// TIA Portal V20 export
FUNCTION_BLOCK "LER_AlignSyncMove"   // FB99, LAD
// stored: Access Published, MemoryReserve 100, SetENOAutomatically false
   VAR_INPUT
      enable : Bool;
      Anode : Bool;
      Cathode : Bool;
      AxisXHomePos { ExternalAccessible := 'False'; ExternalVisible := 'False'; ExternalWritable := 'False'} : LReal;
      AxisY1HomePos { ExternalAccessible := 'False'; ExternalVisible := 'False'; ExternalWritable := 'False'} : LReal;
      AxisY2HomePos { ExternalAccessible := 'False'; ExternalVisible := 'False'; ExternalWritable := 'False'} : LReal;
      MoveSpeed : LReal;
   END_VAR
   VAR_OUTPUT
      error : Bool;
      busy : Bool;
      done : Bool;
      status : Word;
   END_VAR
   VAR_IN_OUT
      moduleInterface : "LER_typeAlignSyncMoveInterface";
      AlignTableAxisX : DB_ANY;
      AlignTableAxisY1 : DB_ANY;
      AlignTableAxisY2 : DB_ANY;
   END_VAR
   VAR
      statMoveRad : LReal;
      statThetaX_Rad : LReal;
      statThetaY1_Rad : LReal;
      statThetaY2_Rad : LReal;
      statDetlaX : LReal;
      statDetlaY1 : LReal;
      statDetlaY2 : LReal;
      instAlignTableAxisXMCMoveAbs : MC_MOVEABSOLUTE;
      instAlignTableAxisY1MCMoveAbs { S7_SetPoint := 'True'} : MC_MOVEABSOLUTE;
      instAlignTableAxisY2MCMoveAbs { S7_SetPoint := 'True'} : MC_MOVEABSOLUTE;
      statPulse { S7_SetPoint := 'True'} : Array[1..50] of Bool;
      statMoveXCmd : Array[1..10] of Bool;
      statMoveY1Cmd : Array[1..10] of Bool;
      statMoveY2Cmd : Array[1..10] of Bool;
   END_VAR
   VAR_TEMP
      tempAlignTableAxisX : REF_TO TO_SynchronousAxis;
      tempAlignTableAxisY1 : REF_TO TO_SynchronousAxis;
      tempAlignTableAxisY2 : REF_TO TO_SynchronousAxis;
   END_VAR
   VAR CONSTANT
      PI : LReal := 3.14159265358979;
      INITIAL_RAD : LReal := 0.0;
      CENTERRADIUS : LReal := 120.0;
   END_VAR
   VAR_TEMP   // added for the SCL form of the ladder/FBD networks
      _w1 : Bool;
   END_VAR
BEGIN

REGION Network 1 (SCL): Axis Config
   #tempAlignTableAxisY1 ?= #AlignTableAxisY1;
   #tempAlignTableAxisY2 ?= #AlignTableAxisY2;
   // #tempAlignTableAxisX ?= #AlignTableAxisX;
END_REGION

REGION Network 2: Error Check
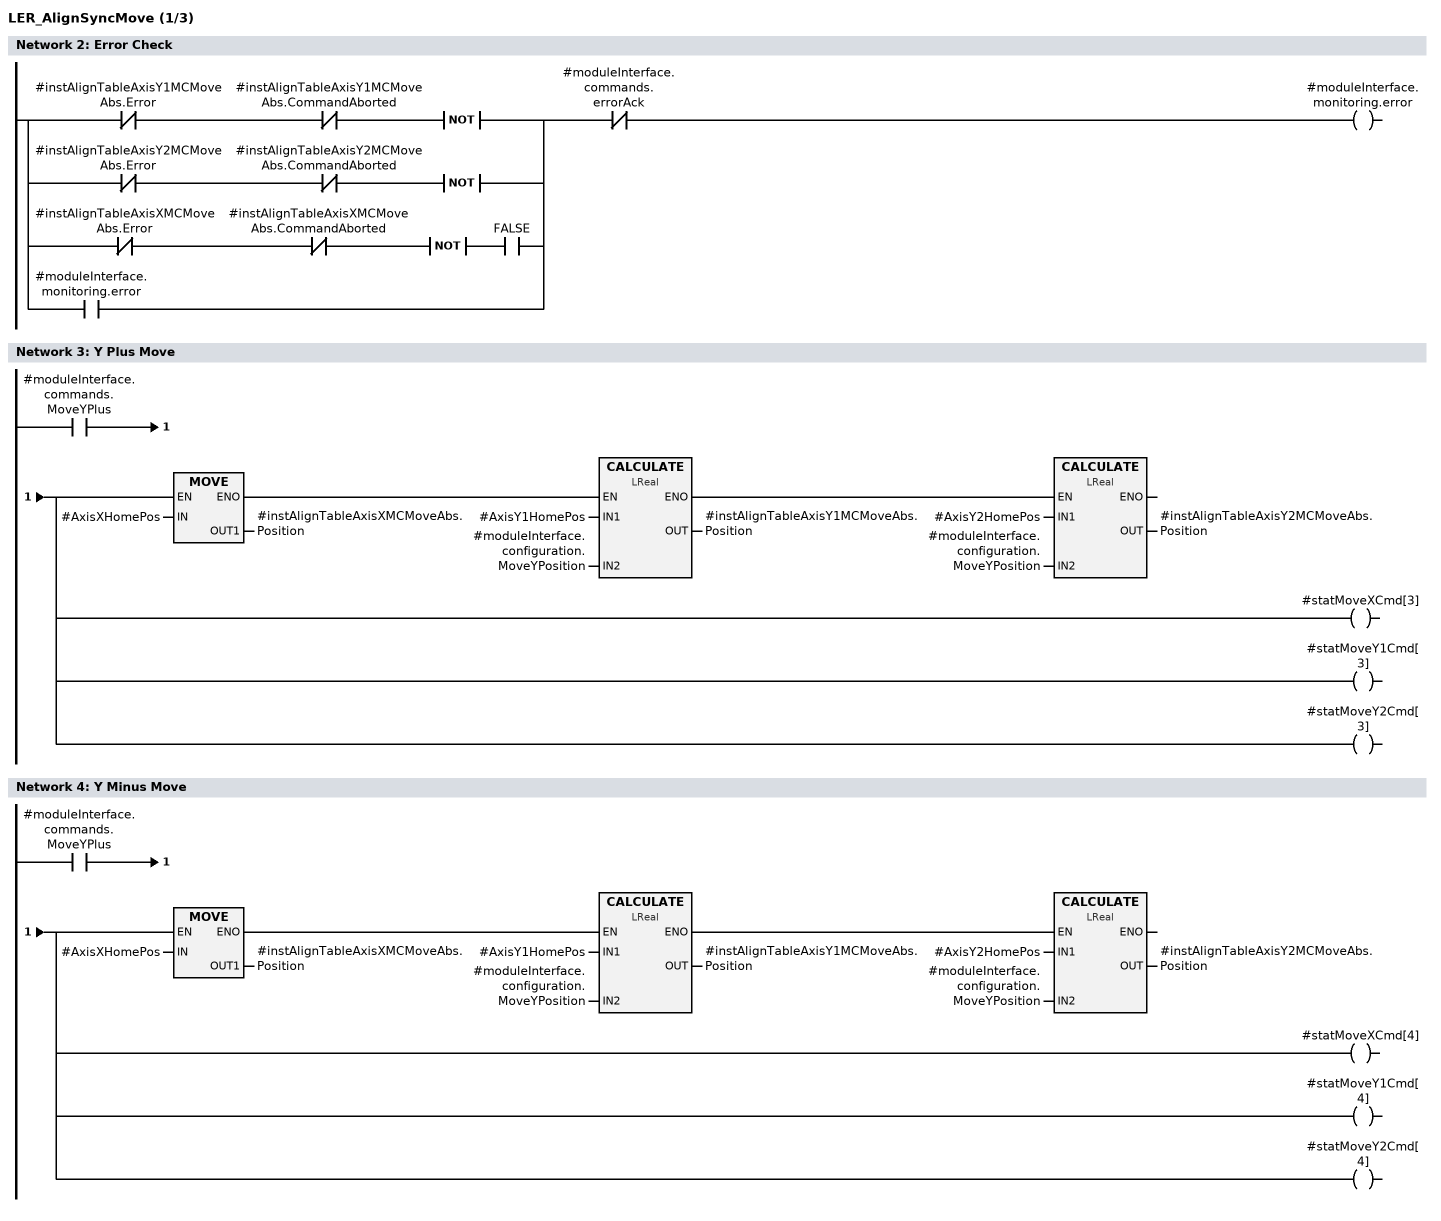
   RUNG wire#powerrail
      I_Contact( #instAlignTableAxisY1MCMoveAbs.Error )
      I_Contact( #instAlignTableAxisY1MCMoveAbs.CommandAborted )
      Not()
      wire#w1
      I_Contact( #moduleInterface.commands.errorAck )
      Coil( #moduleInterface.monitoring.error )
   END_RUNG
   RUNG wire#powerrail
      I_Contact( #instAlignTableAxisY2MCMoveAbs.Error )
      I_Contact( #instAlignTableAxisY2MCMoveAbs.CommandAborted )
      Not()
   END_RUNG wire#w1
   RUNG wire#powerrail
      I_Contact( #instAlignTableAxisXMCMoveAbs.Error )
      I_Contact( #instAlignTableAxisXMCMoveAbs.CommandAborted )
      Not()
      Contact( FALSE )
   END_RUNG wire#w1
   RUNG wire#powerrail
      Contact( #moduleInterface.monitoring.error )
   END_RUNG wire#w1
   // the same network as SCL:
   #moduleInterface.monitoring.error := (NOT (NOT #instAlignTableAxisY1MCMoveAbs.Error AND NOT #instAlignTableAxisY1MCMoveAbs.CommandAborted) OR NOT (NOT #instAlignTableAxisY2MCMoveAbs.Error AND NOT #instAlignTableAxisY2MCMoveAbs.CommandAborted) OR (NOT (NOT #instAlignTableAxisXMCMoveAbs.Error AND NOT #instAlignTableAxisXMCMoveAbs.CommandAborted) AND FALSE) OR #moduleInterface.monitoring.error) AND NOT #moduleInterface.commands.errorAck;
END_REGION

REGION Network 3: Y Plus Move
   RUNG wire#powerrail
      Contact( #moduleInterface.commands.MoveYPlus )
      wire#w1
      Move(in := #AxisXHomePos, out1 => #instAlignTableAxisXMCMoveAbs.Position)
      { S7_Templates := "SrcType := LReal"; S7_Expression := "IN1+IN2" } Calculate(in1 := #AxisY1HomePos, in2 := #moduleInterface.configuration.MoveYPosition, out => #instAlignTableAxisY1MCMoveAbs.Position)
      { S7_Templates := "SrcType := LReal"; S7_Expression := "IN1-IN2" } Calculate(in1 := #AxisY2HomePos, in2 := #moduleInterface.configuration.MoveYPosition, out => #instAlignTableAxisY2MCMoveAbs.Position)
   END_RUNG
   RUNG wire#w1
      Coil( #statMoveXCmd[3] )
   END_RUNG
   RUNG wire#w1
      Coil( #statMoveY1Cmd[3] )
   END_RUNG
   RUNG wire#w1
      Coil( #statMoveY2Cmd[3] )
   END_RUNG
   // the same network as SCL:
   IF #moduleInterface.commands.MoveYPlus THEN
       #instAlignTableAxisXMCMoveAbs.Position := #AxisXHomePos;
       #instAlignTableAxisY1MCMoveAbs.Position := #AxisY1HomePos+#moduleInterface.configuration.MoveYPosition;
       #instAlignTableAxisY2MCMoveAbs.Position := #AxisY2HomePos-#moduleInterface.configuration.MoveYPosition;
   END_IF;
   #statMoveXCmd[3] := #moduleInterface.commands.MoveYPlus;
   #statMoveY1Cmd[3] := #moduleInterface.commands.MoveYPlus;
   #statMoveY2Cmd[3] := #moduleInterface.commands.MoveYPlus;
END_REGION

REGION Network 4: Y Minus Move
   RUNG wire#powerrail
      Contact( #moduleInterface.commands.MoveYPlus )
      wire#w1
      Move(in := #AxisXHomePos, out1 => #instAlignTableAxisXMCMoveAbs.Position)
      { S7_Templates := "SrcType := LReal"; S7_Expression := "IN1-IN2" } Calculate(in1 := #AxisY1HomePos, in2 := #moduleInterface.configuration.MoveYPosition, out => #instAlignTableAxisY1MCMoveAbs.Position)
      { S7_Templates := "SrcType := LReal"; S7_Expression := "IN1+IN2" } Calculate(in1 := #AxisY2HomePos, in2 := #moduleInterface.configuration.MoveYPosition, out => #instAlignTableAxisY2MCMoveAbs.Position)
   END_RUNG
   RUNG wire#w1
      Coil( #statMoveXCmd[4] )
   END_RUNG
   RUNG wire#w1
      Coil( #statMoveY1Cmd[4] )
   END_RUNG
   RUNG wire#w1
      Coil( #statMoveY2Cmd[4] )
   END_RUNG
   // the same network as SCL:
   IF #moduleInterface.commands.MoveYPlus THEN
       #instAlignTableAxisXMCMoveAbs.Position := #AxisXHomePos;
       #instAlignTableAxisY1MCMoveAbs.Position := #AxisY1HomePos-#moduleInterface.configuration.MoveYPosition;
       #instAlignTableAxisY2MCMoveAbs.Position := #AxisY2HomePos+#moduleInterface.configuration.MoveYPosition;
   END_IF;
   #statMoveXCmd[4] := #moduleInterface.commands.MoveYPlus;
   #statMoveY1Cmd[4] := #moduleInterface.commands.MoveYPlus;
   #statMoveY2Cmd[4] := #moduleInterface.commands.MoveYPlus;
END_REGION

REGION Network 5: Mapping Cmd
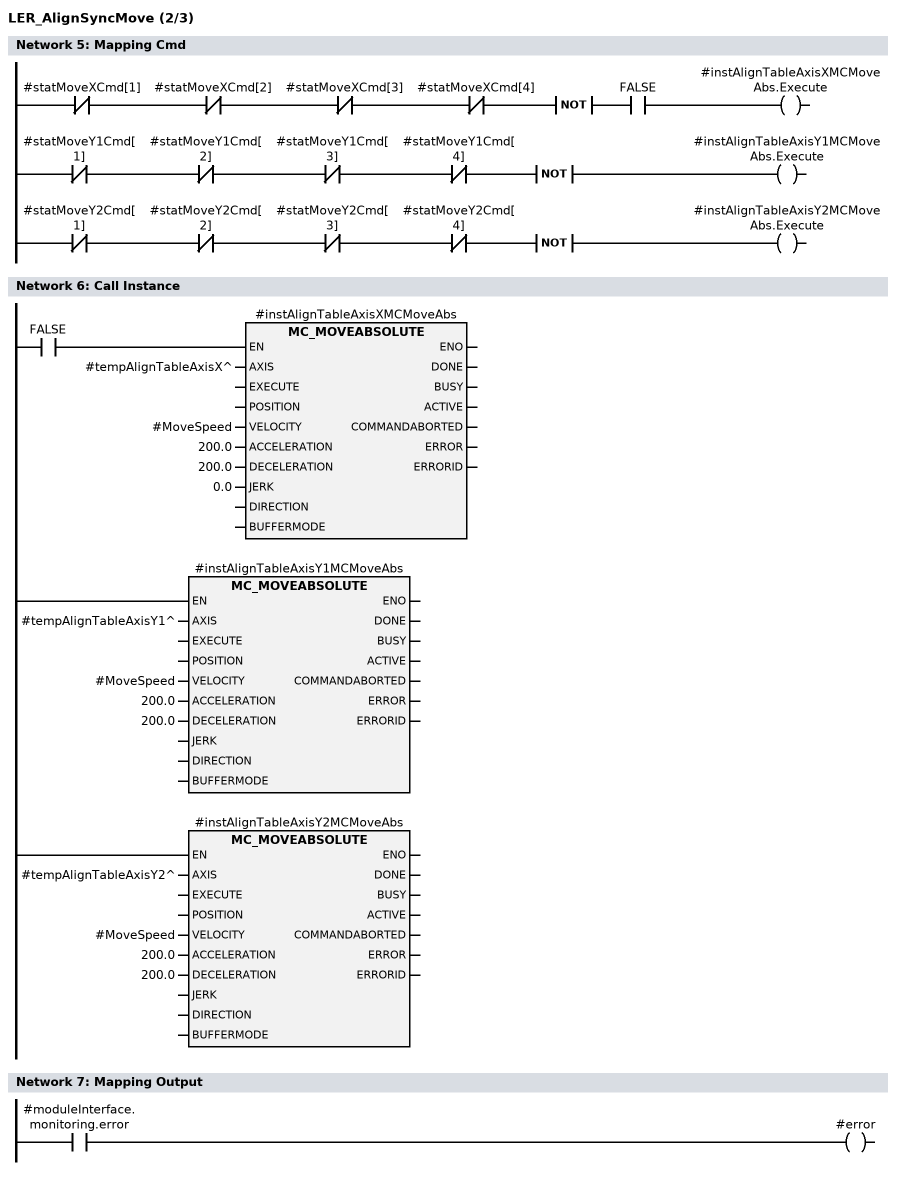
   RUNG wire#powerrail
      I_Contact( #statMoveXCmd[1] )
      I_Contact( #statMoveXCmd[2] )
      I_Contact( #statMoveXCmd[3] )
      I_Contact( #statMoveXCmd[4] )
      Not()
      Contact( FALSE )
      Coil( #instAlignTableAxisXMCMoveAbs.Execute )
   END_RUNG
   RUNG wire#powerrail
      I_Contact( #statMoveY1Cmd[1] )
      I_Contact( #statMoveY1Cmd[2] )
      I_Contact( #statMoveY1Cmd[3] )
      I_Contact( #statMoveY1Cmd[4] )
      Not()
      Coil( #instAlignTableAxisY1MCMoveAbs.Execute )
   END_RUNG
   RUNG wire#powerrail
      I_Contact( #statMoveY2Cmd[1] )
      I_Contact( #statMoveY2Cmd[2] )
      I_Contact( #statMoveY2Cmd[3] )
      I_Contact( #statMoveY2Cmd[4] )
      Not()
      Coil( #instAlignTableAxisY2MCMoveAbs.Execute )
   END_RUNG
   // the same network as SCL:
   #instAlignTableAxisXMCMoveAbs.Execute := NOT (NOT #statMoveXCmd[1] AND NOT #statMoveXCmd[2] AND NOT #statMoveXCmd[3] AND NOT #statMoveXCmd[4]) AND FALSE;
   #instAlignTableAxisY1MCMoveAbs.Execute := NOT (NOT #statMoveY1Cmd[1] AND NOT #statMoveY1Cmd[2] AND NOT #statMoveY1Cmd[3] AND NOT #statMoveY1Cmd[4]);
   #instAlignTableAxisY2MCMoveAbs.Execute := NOT (NOT #statMoveY2Cmd[1] AND NOT #statMoveY2Cmd[2] AND NOT #statMoveY2Cmd[3] AND NOT #statMoveY2Cmd[4]);
END_REGION

REGION Network 6: Call Instance
   RUNG wire#powerrail
      Contact( FALSE )
      #instAlignTableAxisXMCMoveAbs.MC_MOVEABSOLUTE(Axis := #tempAlignTableAxisX^, Execute :=, Position :=, Velocity := #MoveSpeed, Acceleration := 200.0, Deceleration := 200.0, Jerk := 0.0, Direction :=, BufferMode :=, Done =>, Busy =>, Active =>, CommandAborted =>, Error =>, ErrorId =>)
   END_RUNG
   RUNG wire#powerrail
      #instAlignTableAxisY1MCMoveAbs.MC_MOVEABSOLUTE(Axis := #tempAlignTableAxisY1^, Execute :=, Position :=, Velocity := #MoveSpeed, Acceleration := 200.0, Deceleration := 200.0, Jerk :=, Direction :=, BufferMode :=, Done =>, Busy =>, Active =>, CommandAborted =>, Error =>, ErrorId =>)
   END_RUNG
   RUNG wire#powerrail
      #instAlignTableAxisY2MCMoveAbs.MC_MOVEABSOLUTE(Axis := #tempAlignTableAxisY2^, Execute :=, Position :=, Velocity := #MoveSpeed, Acceleration := 200.0, Deceleration := 200.0, Jerk :=, Direction :=, BufferMode :=, Done =>, Busy =>, Active =>, CommandAborted =>, Error =>, ErrorId =>)
   END_RUNG
   // the same network as SCL:
   IF FALSE THEN
       #instAlignTableAxisXMCMoveAbs(Axis := #tempAlignTableAxisX^,   // MC_MOVEABSOLUTE
                               Velocity := #MoveSpeed,
                               Acceleration := 200.0,
                               Deceleration := 200.0,
                               Jerk := 0.0);
   END_IF;
   #instAlignTableAxisY1MCMoveAbs(Axis := #tempAlignTableAxisY1^,   // MC_MOVEABSOLUTE
                           Velocity := #MoveSpeed,
                           Acceleration := 200.0,
                           Deceleration := 200.0);
   #instAlignTableAxisY2MCMoveAbs(Axis := #tempAlignTableAxisY2^,   // MC_MOVEABSOLUTE
                           Velocity := #MoveSpeed,
                           Acceleration := 200.0,
                           Deceleration := 200.0);
END_REGION

REGION Network 7: Mapping Output
   RUNG wire#powerrail
      Contact( #moduleInterface.monitoring.error )
      Coil( #error )
   END_RUNG
   // the same network as SCL:
   #error := #moduleInterface.monitoring.error;
END_REGION

REGION Network 8: ******************** Unused ********************
END_REGION

REGION Network 9 (SCL): [Unused] CalCulate Axis Distance[mm]/Deg
   // 아래 연산식은 설비사로 부터 받은 계산식으로 연산하였습니다. 연산 이상 시, 설비사에게 계산식을 새로 받아야합니다.

   // REGION 이동 각도 변환 (Deg -> Rad)
   //     IF #moduleInterface.commands.MoveCw THEN
   //         #statMoveRad := - #moduleInterface.configuration.MoveDeg * (#PI / 180.0);
   //     ELSIF #moduleInterface.commands.MoveCcw THEN
   //         #statMoveRad := #moduleInterface.configuration.MoveDeg * (#PI / 180.0);
   //     END_IF;
   // END_REGION

   // REGION 모터 중심 각도 Rad 연산
   //     #statThetaX_Rad := 180.0 * (#PI / 180.0);
   //     #statThetaY1_Rad := 90.0 * (#PI / 180.0);
   //     #statThetaY2_Rad := 270.0 * (#PI / 180.0);
   // END_REGION

   // REGION Deg 이동량을 축당 mm 이동량 산출
   //     #statDetlaX := #CENTERRADIUS * SIN(#statMoveRad + #statThetaX_Rad + #INITIAL_RAD) - #CENTERRADIUS * SIN(#statThetaX_Rad + #INITIAL_RAD);
   //     #statDetlaY1 := #CENTERRADIUS * COS(#statMoveRad + #statThetaY1_Rad + #INITIAL_RAD) - #CENTERRADIUS * COS(#statThetaY1_Rad + #INITIAL_RAD);
   //     #statDetlaY2 := #CENTERRADIUS * COS(#statMoveRad + #statThetaY2_Rad + #INITIAL_RAD) - #CENTERRADIUS * COS(#statThetaY2_Rad + #INITIAL_RAD);
   // END_REGION
END_REGION

REGION Network 10: [Unused] Deg CW Move
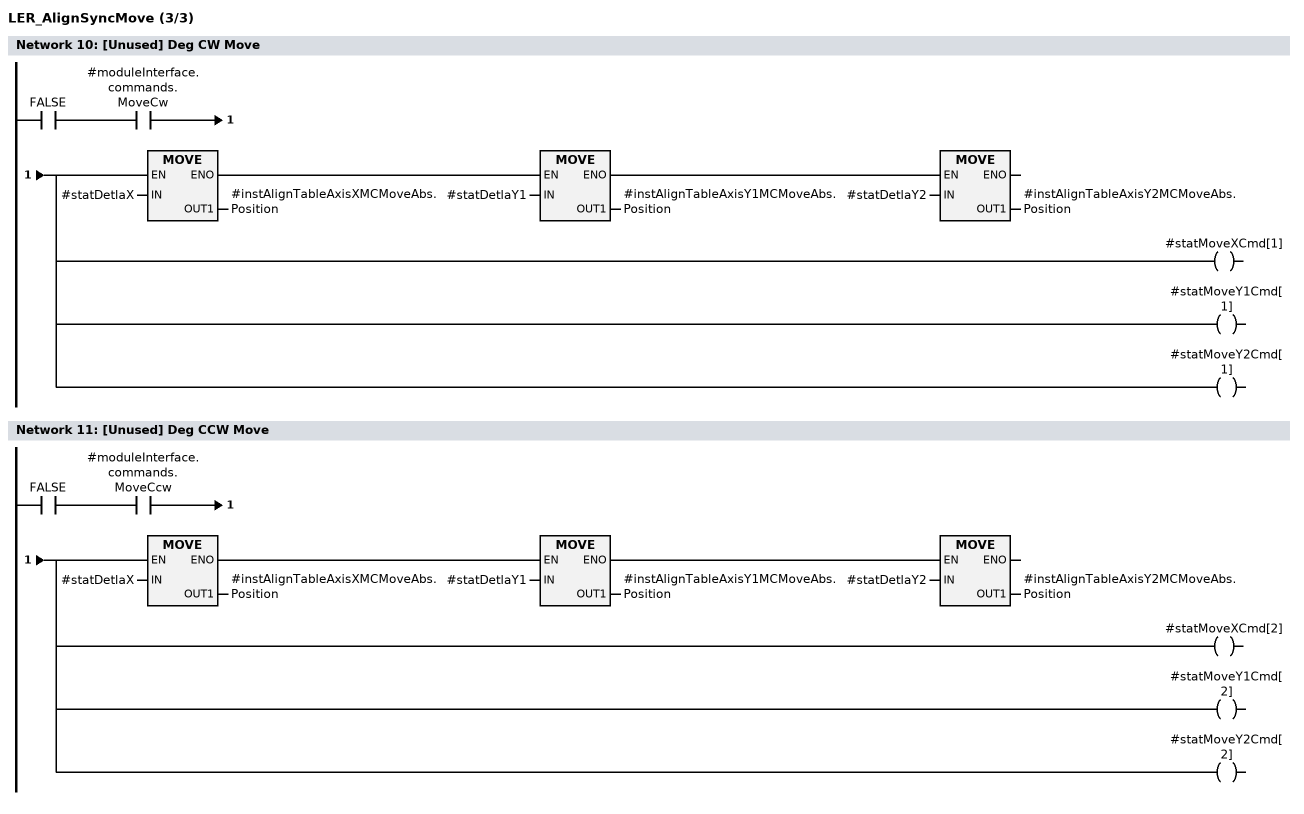
   RUNG wire#powerrail
      Contact( FALSE )
      Contact( #moduleInterface.commands.MoveCw )
      wire#w1
      Move(in := #statDetlaX, out1 => #instAlignTableAxisXMCMoveAbs.Position)
      Move(in := #statDetlaY1, out1 => #instAlignTableAxisY1MCMoveAbs.Position)
      Move(in := #statDetlaY2, out1 => #instAlignTableAxisY2MCMoveAbs.Position)
   END_RUNG
   RUNG wire#w1
      Coil( #statMoveXCmd[1] )
   END_RUNG
   RUNG wire#w1
      Coil( #statMoveY1Cmd[1] )
   END_RUNG
   RUNG wire#w1
      Coil( #statMoveY2Cmd[1] )
   END_RUNG
   // the same network as SCL:
   #_w1 := FALSE AND #moduleInterface.commands.MoveCw;
   IF #_w1 THEN
       #instAlignTableAxisXMCMoveAbs.Position := #statDetlaX;
       #instAlignTableAxisY1MCMoveAbs.Position := #statDetlaY1;
       #instAlignTableAxisY2MCMoveAbs.Position := #statDetlaY2;
   END_IF;
   #statMoveXCmd[1] := #_w1;
   #statMoveY1Cmd[1] := #_w1;
   #statMoveY2Cmd[1] := #_w1;
END_REGION

REGION Network 11: [Unused] Deg CCW Move
   RUNG wire#powerrail
      Contact( FALSE )
      Contact( #moduleInterface.commands.MoveCcw )
      wire#w1
      Move(in := #statDetlaX, out1 => #instAlignTableAxisXMCMoveAbs.Position)
      Move(in := #statDetlaY1, out1 => #instAlignTableAxisY1MCMoveAbs.Position)
      Move(in := #statDetlaY2, out1 => #instAlignTableAxisY2MCMoveAbs.Position)
   END_RUNG
   RUNG wire#w1
      Coil( #statMoveXCmd[2] )
   END_RUNG
   RUNG wire#w1
      Coil( #statMoveY1Cmd[2] )
   END_RUNG
   RUNG wire#w1
      Coil( #statMoveY2Cmd[2] )
   END_RUNG
   // the same network as SCL:
   #_w1 := FALSE AND #moduleInterface.commands.MoveCcw;
   IF #_w1 THEN
       #instAlignTableAxisXMCMoveAbs.Position := #statDetlaX;
       #instAlignTableAxisY1MCMoveAbs.Position := #statDetlaY1;
       #instAlignTableAxisY2MCMoveAbs.Position := #statDetlaY2;
   END_IF;
   #statMoveXCmd[2] := #_w1;
   #statMoveY1Cmd[2] := #_w1;
   #statMoveY2Cmd[2] := #_w1;
END_REGION
END_FUNCTION_BLOCK
